// TIA Portal V20 export
FUNCTION_BLOCK "FB_IO_Device_Production_And_Rework"   // FB5, LAD
{ S7_Optimized_Access := 'TRUE' }
// stored: MemoryReserve 100, SetENOAutomatically false
   VAR_INPUT
      Start : Bool;
      Manual_Turn_On_Motor_Caroussel : Bool;
      Manual_Turn_On_Motor_Conveyor_Belt : Bool;
      Water_Foutain_Fail_Functional_Test : Bool;
      Select_Motor_Speed : SInt;
      Carousel_Voltage_Selection : SInt;
      In_PLC_Production_And_Rework : "IO_Device_Conveyor_Belt_Input";
   END_VAR
   VAR_OUTPUT
      Comunication_Error : Bool;
      Emergency_Stop_Release : Bool;
      Trigger_Read_Serial_Number_Entrace_Functional_Test : Bool;
      Trigger_Read_Serial_Number_Exit_Functional_Test : Bool;
      Selected_Voltage_220V : Bool;
      Selected_Voltage_127V : Bool;
      Carousel_Frequency_Inverter_Fail : Bool;
      Conveyor_Belt_Functional_Test_Inverter_Fail : Bool;
      Out_PLC_Production_And_Rework : "IO_Device_Conveyor_Belt_Ouput";
   END_VAR
   VAR
      Timer_Alarme_A_1 { S7_SetPoint := 'True'} : TON_TIME;
      Timer_Alarme_B_1 { S7_SetPoint := 'True'} : TON_TIME;
   END_VAR
BEGIN

REGION Network 1
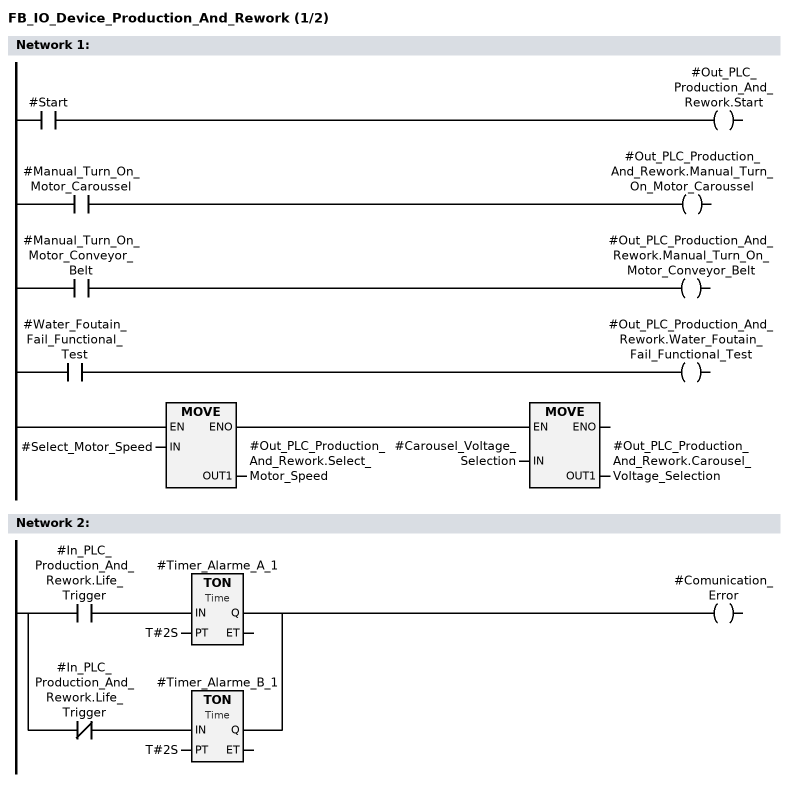
   RUNG wire#powerrail
      Contact( #Start )
      Coil( #Out_PLC_Production_And_Rework.Start )
   END_RUNG
   RUNG wire#powerrail
      Contact( #Manual_Turn_On_Motor_Caroussel )
      Coil( #Out_PLC_Production_And_Rework.Manual_Turn_On_Motor_Caroussel )
   END_RUNG
   RUNG wire#powerrail
      Contact( #Manual_Turn_On_Motor_Conveyor_Belt )
      Coil( #Out_PLC_Production_And_Rework.Manual_Turn_On_Motor_Conveyor_Belt )
   END_RUNG
   RUNG wire#powerrail
      Contact( #Water_Foutain_Fail_Functional_Test )
      Coil( #Out_PLC_Production_And_Rework.Water_Foutain_Fail_Functional_Test )
   END_RUNG
   RUNG wire#powerrail
      Move(in := #Select_Motor_Speed, out1 => #Out_PLC_Production_And_Rework.Select_Motor_Speed)
      Move(in := #Carousel_Voltage_Selection, out1 => #Out_PLC_Production_And_Rework.Carousel_Voltage_Selection)
   END_RUNG
   // the same network as SCL:
   #Out_PLC_Production_And_Rework.Start := #Start;
   #Out_PLC_Production_And_Rework.Manual_Turn_On_Motor_Caroussel := #Manual_Turn_On_Motor_Caroussel;
   #Out_PLC_Production_And_Rework.Manual_Turn_On_Motor_Conveyor_Belt := #Manual_Turn_On_Motor_Conveyor_Belt;
   #Out_PLC_Production_And_Rework.Water_Foutain_Fail_Functional_Test := #Water_Foutain_Fail_Functional_Test;
   #Out_PLC_Production_And_Rework.Select_Motor_Speed := #Select_Motor_Speed;
   #Out_PLC_Production_And_Rework.Carousel_Voltage_Selection := #Carousel_Voltage_Selection;
END_REGION

REGION Network 2
   RUNG wire#powerrail
      Contact( #In_PLC_Production_And_Rework.Life_Trigger )
      { S7_Templates := "time_type := Time" } #Timer_Alarme_A_1.TON(pt := T#2S, et =>)
      wire#w1
      Coil( #Comunication_Error )
   END_RUNG
   RUNG wire#powerrail
      I_Contact( #In_PLC_Production_And_Rework.Life_Trigger )
      { S7_Templates := "time_type := Time" } #Timer_Alarme_B_1.TON(pt := T#2S, et =>)
   END_RUNG wire#w1
   // the same network as SCL:
   #Timer_Alarme_A_1(IN := #In_PLC_Production_And_Rework.Life_Trigger, PT := T#2S);   // TON
   #Timer_Alarme_B_1(IN := NOT #In_PLC_Production_And_Rework.Life_Trigger, PT := T#2S);   // TON
   #Comunication_Error := #Timer_Alarme_A_1.Q OR #Timer_Alarme_B_1.Q;
END_REGION

REGION Network 3
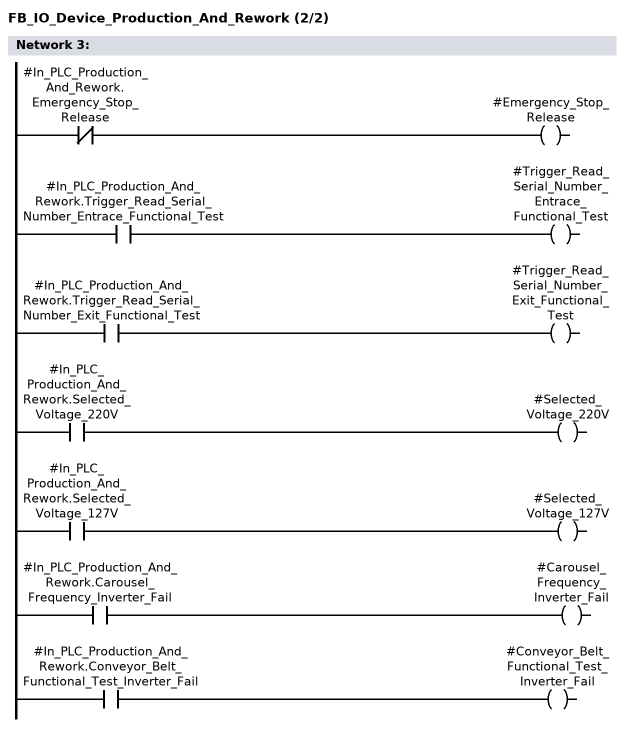
   RUNG wire#powerrail
      I_Contact( #In_PLC_Production_And_Rework.Emergency_Stop_Release )
      Coil( #Emergency_Stop_Release )
   END_RUNG
   RUNG wire#powerrail
      Contact( #In_PLC_Production_And_Rework.Trigger_Read_Serial_Number_Entrace_Functional_Test )
      Coil( #Trigger_Read_Serial_Number_Entrace_Functional_Test )
   END_RUNG
   RUNG wire#powerrail
      Contact( #In_PLC_Production_And_Rework.Trigger_Read_Serial_Number_Exit_Functional_Test )
      Coil( #Trigger_Read_Serial_Number_Exit_Functional_Test )
   END_RUNG
   RUNG wire#powerrail
      Contact( #In_PLC_Production_And_Rework.Selected_Voltage_220V )
      Coil( #Selected_Voltage_220V )
   END_RUNG
   RUNG wire#powerrail
      Contact( #In_PLC_Production_And_Rework.Selected_Voltage_127V )
      Coil( #Selected_Voltage_127V )
   END_RUNG
   RUNG wire#powerrail
      Contact( #In_PLC_Production_And_Rework.Carousel_Frequency_Inverter_Fail )
      Coil( #Carousel_Frequency_Inverter_Fail )
   END_RUNG
   RUNG wire#powerrail
      Contact( #In_PLC_Production_And_Rework.Conveyor_Belt_Functional_Test_Inverter_Fail )
      Coil( #Conveyor_Belt_Functional_Test_Inverter_Fail )
   END_RUNG
   // the same network as SCL:
   #Emergency_Stop_Release := NOT #In_PLC_Production_And_Rework.Emergency_Stop_Release;
   #Trigger_Read_Serial_Number_Entrace_Functional_Test := #In_PLC_Production_And_Rework.Trigger_Read_Serial_Number_Entrace_Functional_Test;
   #Trigger_Read_Serial_Number_Exit_Functional_Test := #In_PLC_Production_And_Rework.Trigger_Read_Serial_Number_Exit_Functional_Test;
   #Selected_Voltage_220V := #In_PLC_Production_And_Rework.Selected_Voltage_220V;
   #Selected_Voltage_127V := #In_PLC_Production_And_Rework.Selected_Voltage_127V;
   #Carousel_Frequency_Inverter_Fail := #In_PLC_Production_And_Rework.Carousel_Frequency_Inverter_Fail;
   #Conveyor_Belt_Functional_Test_Inverter_Fail := #In_PLC_Production_And_Rework.Conveyor_Belt_Functional_Test_Inverter_Fail;
END_REGION
END_FUNCTION_BLOCK
